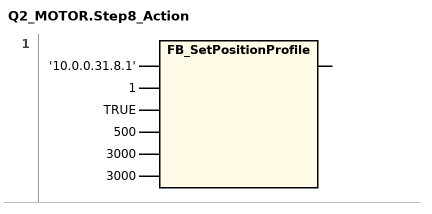
// NETWORK 1
FB_SetPositionProfile('10.0.0.31.8.1', 1, TRUE, 500, 3000, 3000);
END_ACTION

END_PROGRAM

// ---- POUs/testop.TcPOU
PROGRAM testop
VAR
	TP_OP: TON;
	START: BOOL:=FALSE;
	TP_OP2: TON;
END_VAR



IF(GEMMA.STEP='F1') AND RUN_CG THEN

IF(NOT(TP_OP.Q ) AND NOT(TP_OP2.Q)) THEN
START:=TRUE;
ELSIF(TP_OP.Q AND TP_OP2.Q) THEN
START:=FALSE;
END_IF

TP_OP(IN:= START, PT:= CG_DELAY);

TP_OP2(IN:= TP_OP.Q, PT:= T#30s);

VAC_DO.WAGON_OPERATOR1:= NOT(TP_OP.Q);

VAC_DO.WAGON_OPERATOR2:=FALSE;


END_IF
;

END_PROGRAM

// ---- POUs/CHECK_VALVES_SENSORS.TcPOU
FUNCTION_BLOCK CHECK_VALVES_SENSORS
VAR_INPUT
END_VAR
VAR_OUTPUT
END_VAR
VAR
	STEP: INT := 0;
END_VAR

(**************************************************************
*
*
* Check Valves sensors
*
*
***************************************************************)
CASE STEP OF

0: (*Init*)
	STEP := STEP+1;

1: (*Initialise valves and variables*)
;
ELSE
    ;
END_CASE;

END_FUNCTION_BLOCK

// ---- POUs/EVENTS.TcPOU
PROGRAM EVENTS
VAR
END_VAR

LogEvent_1000_1 (SourceID := 1000,EventID := 1,bSetEvent := bSetEvent_1000_1, bQuit := bQuitEvent_1000_1);
LogEvent_1000_2 (SourceID := 1000,EventID := 2,bSetEvent := bSetEvent_1000_2, bQuit := bQuitEvent_1000_2);

END_PROGRAM

// ---- GlobalTextList.TcGTLO
TEXTLIST GlobalTextList
  23 = '%0.1f bar'
  25 = '%0.1f mA'
  24 = '%0.1f ml/min'
  22 = '%d'
  21 = '%s'
  5 = 'AIR'
  16 = 'ASK_RELEASE_OP1'
  17 = 'ASK_RELEASE_OP2'
  19 = 'AUTO'
  6 = 'CONVEYOR'
  12 = 'DOORS_OPEN'
  14 = 'INIT_OK'
  20 = 'MANUEL'
  10 = 'PMAX_RELEASE'
  3 = 'PMAX_STATUS'
  11 = 'PRINT_RELEASE'
  4 = 'PRINT_STATUS'
  1 = 'Q1_STATUS'
  8 = 'Q1__RELEASE'
  9 = 'Q2_RELEASE'
  2 = 'Q2_STATUS'
  15 = 'SAFETY_OK'
  18 = 'SAFETY_RESET'
  13 = 'TIMOUT_TANK_VAC'
  7 = 'VAC_RELEASE'
  0 = 'VAC_STATUS'
END_TEXTLIST

// ---- Visualizations/FLAGS.TcVIS
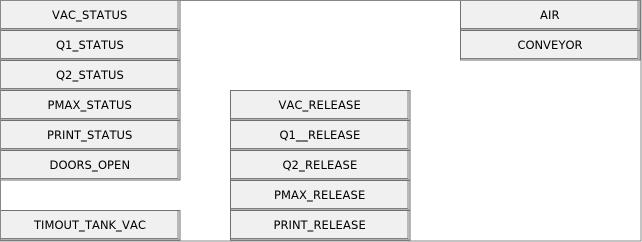
VISUALIZATION FLAGS  // 642x242
    Button (0,0 180x30), "VAC_STATUS", pressed state: Flag_Variables.FLAGS .VAC_STATUS
        toggle Flag_Variables.FLAGS .VAC_STATUS
    Button (0,30 180x30), "Q1_STATUS", pressed state: Flag_Variables.FLAGS .Q1_STATUS
        toggle Flag_Variables.FLAGS .Q1_STATUS
    Button (0,60 180x30), "Q2_STATUS", pressed state: Flag_Variables.FLAGS .Q2_STATUS
        toggle Flag_Variables.FLAGS .Q2_STATUS
    Button (0,90 180x30), "PMAX_STATUS", pressed state: Flag_Variables.FLAGS .PMAX_STATUS
        toggle Flag_Variables.FLAGS .PMAX_STATUS
    Button (0,120 180x30), "PRINT_STATUS", pressed state: Flag_Variables.FLAGS .PRINT_STATUS
        toggle Flag_Variables.FLAGS .PRINT_STATUS
    Button (460,0 180x30), "AIR", pressed state: IOs_Variables.VAC_DO .AIR_VALVE
        toggle IOs_Variables.VAC_DO .AIR_VALVE
    Button (460,30 180x30), "CONVEYOR", pressed state: IOs_Variables.POW_DO .CONVEYOR_RELAIS
        toggle IOs_Variables.POW_DO .CONVEYOR_RELAIS
    Button (230,90 180x30), "VAC_RELEASE", pressed state: Flag_Variables.FLAGS .VAC_RELEASE_CARRIER
        toggle Flag_Variables.FLAGS .VAC_RELEASE_CARRIER
    Button (230,120 180x30), "Q1__RELEASE", pressed state: Flag_Variables.FLAGS .Q1_RELEASE_CARRIER
        toggle Flag_Variables.FLAGS .Q1_RELEASE_CARRIER
    Button (230,150 180x30), "Q2_RELEASE", pressed state: Flag_Variables.FLAGS .Q2_RELEASE_CARRIER
        toggle Flag_Variables.FLAGS .Q2_RELEASE_CARRIER
    Button (230,180 180x30), "PMAX_RELEASE", pressed state: Flag_Variables.FLAGS .PMAX_RELEASE_CARRIER
        toggle Flag_Variables.FLAGS .PMAX_RELEASE_CARRIER
    Button (230,210 180x30), "PRINT_RELEASE", pressed state: Flag_Variables.FLAGS .PRINT_RELEASE_CARRIER
        toggle Flag_Variables.FLAGS .PRINT_RELEASE_CARRIER
    Button (0,150 180x30), "DOORS_OPEN", pressed state: Flag_Variables.FLAGS .DOORS_OPEN
        toggle Flag_Variables.FLAGS .DOORS_OPEN
    Button (0,210 180x30), "TIMOUT_TANK_VAC", pressed state: WATER_TANKS.TIMOUT_TANK_VAC
        toggle WATER_TANKS.TIMOUT_TANK_VAC
END_VISUALIZATION

// ---- Visualizations/GEMMA.TcVIS
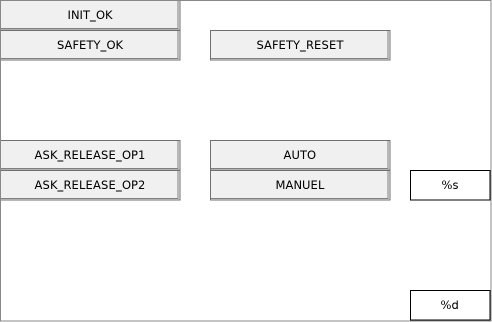
VISUALIZATION GEMMA  // 492x322
    Button (0,0 180x30), "INIT_OK", pressed state: Flag_Variables.FLAGS .INIT_OK
        toggle Flag_Variables.FLAGS .INIT_OK
    Button (0,30 180x30), "SAFETY_OK", pressed state: Flag_Variables.FLAGS .SAFETY_OK
        toggle Flag_Variables.FLAGS .SAFETY_OK
    Button (0,140 180x30), "ASK_RELEASE_OP1", pressed state: IOs_Variables.PRINT_DI .ASK_RELEASE_JIG_OP1
        toggle IOs_Variables.PRINT_DI .ASK_RELEASE_JIG_OP1
    Button (0,170 180x30), "ASK_RELEASE_OP2", pressed state: IOs_Variables.PRINT_DI .ASK_RELEASE_JIG_OP2
        toggle IOs_Variables.PRINT_DI .ASK_RELEASE_JIG_OP2
    Button (210,30 180x30), "SAFETY_RESET", pressed state: Flag_Variables.SAFETY_OUT .NOT_AUS_RESET
        toggle Flag_Variables.SAFETY_OUT .NOT_AUS_RESET
    Button (210,140 180x30), "AUTO", pressed state: Flag_Variables.FLAGS .AUTO
        toggle Flag_Variables.FLAGS .AUTO
    Button (210,170 180x30), "MANUEL", pressed state: Flag_Variables.FLAGS .MANUAL
        toggle Flag_Variables.FLAGS .MANUAL
    Rectangle (410,170 80x30), "%s", text variable: GEMMA.STEP
    Rectangle (410,290 80x30), "%d", text variable: LEDS.M1_FB_GetPositionIs.PositionIs
END_VISUALIZATION

// ---- Visualizations/Motor.TcVIS
VISUALIZATION Motor  // 2x2
END_VISUALIZATION

// ---- Visualizations/P_MAX.TcVIS
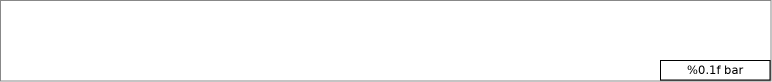
VISUALIZATION P_MAX  // 772x82
    Rectangle (660,60 110x20), "%0.1f bar", text variable: IOs_Variables.PMAX_PRESSURE_LOOSE
END_VISUALIZATION

// ---- Visualizations/Q1.TcVIS
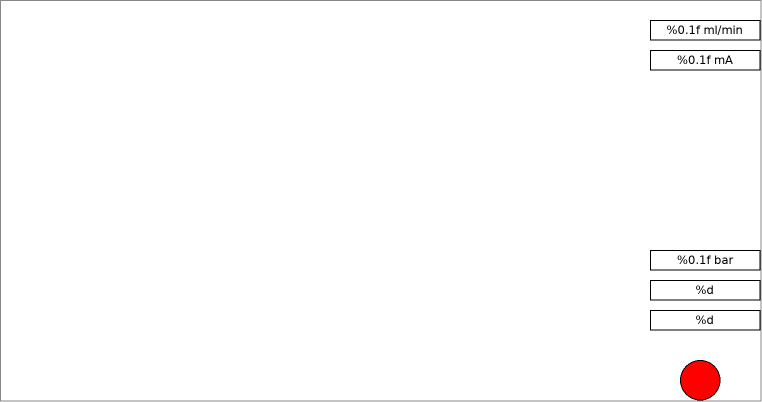
VISUALIZATION Q1  // 762x402
    Rectangle (650,20 110x20), "%0.1f ml/min", text variable: IOs_Variables.Q1_CALCULETED_FLOW
    Rectangle (650,280 110x20), "%d", text variable: LEDS.M1_FB_GetPositionIs.PositionIs
    Rectangle (650,250 110x20), "%0.1f bar", text variable: IOs_Variables.Q1_PRESSURE_SENSOR_VALUE
    Rectangle (650,310 110x20), "%d", text variable: Q1.STEP
    Ellipse (680,360 40x40), colour toggle: (LEDS.M1_FB_GetEnableState.IsEnabled) <> 0
    Rectangle (650,50 110x20), "%0.1f mA", text variable: IOs_Variables.Q1_CURRENT
END_VISUALIZATION

// ---- Visualizations/Q2.TcVIS
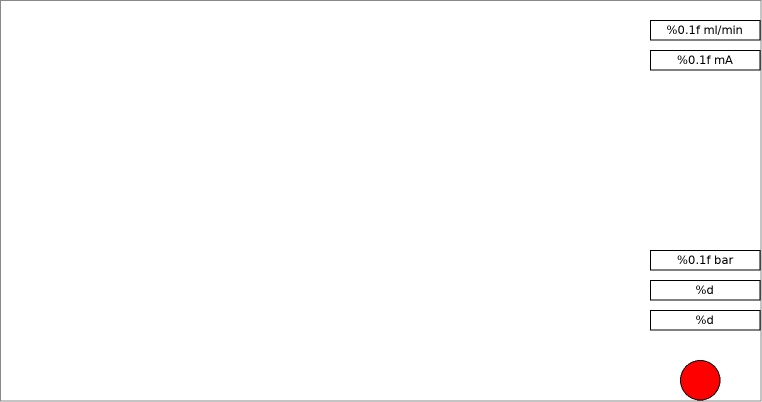
VISUALIZATION Q2  // 762x402
    Rectangle (650,20 110x20), "%0.1f ml/min", text variable: IOs_Variables.Q2_CALCULETED_FLOW
    Rectangle (650,280 110x20), "%d", text variable: LEDS.M2_FB_GetPositionIs.PositionIs
    Rectangle (650,250 110x20), "%0.1f bar", text variable: IOs_Variables.Q2_PRESSURE_SENSOR_VALUE
    Rectangle (650,310 110x20), "%d", text variable: Q2.STEP
    Ellipse (680,360 40x40), colour toggle: (LEDS.M2_FB_GetEnableState.IsEnabled) <> 0
    Rectangle (650,50 110x20), "%0.1f mA", text variable: IOs_Variables.Q2_CURRENT
END_VISUALIZATION

// ---- Visualizations/VAC.TcVIS
VISUALIZATION VAC  // 2x2
END_VISUALIZATION
